FUNCTION Convert_TOD_TO_BOOL : Hresult
VAR_INPUT
	in : TOD;
	out : REFERENCE TO BOOL;
END_VAR
VAR
	converted : BOOL;
END_VAR

converted := TOD_TO_BOOL(in);

IF (BOOL_TO_TOD(converted) <> in) THEN
	Convert_TOD_TO_BOOL := INCOMPATIBLE;
	RETURN;
END_IF

out := converted;

END_FUNCTION

(* stored: Version 1.1.0.1, ProductVersion 3.1.4024.12
   POU Convert_TOD_TO_BOOL: Id {bbf8e7a8-7360-4f12-a692-93de6c6300ae}, SpecialFunc None *)
